// TIA Portal V17 export
// export: Created 2023-02-14T02:49:13.310207Z, ExportSetting WithDefaults, DisplayName Totally Integrated Automation Portal, DisplayVersion V17, DisplayName TIA Portal Openness, DisplayVersion V17, DisplayName TIA Portal Teamcenter Gateway, DisplayVersion V17, DisplayName TIA Portal Version Control Interface, DisplayVersion V17, DisplayName SINAMICS Startdrive Advanced, DisplayVersion V17, DisplayName SINAMICS Startdrive G130, G150, S120, S150, SINAMICS MV, S210, DisplayVersion V17, DisplayName SINAMICS Startdrive G110M, G120, G120C, G120D, G120P, G115D, DisplayVersion V17, DisplayName STEP 7 Professional, DisplayVersion V17, DisplayName STEP 7 Safety, DisplayVersion V17, DisplayName WinCC Professional, DisplayVersion V17
DATA_BLOCK "Mix_to_Salt"   // DB20
{ S7_Optimized_Access := 'FALSE' }
VERSION : 0.1
// stored: AutoNumber false, DBAccessibleFromOPCUA true, DBAccessibleFromWebserver true, IsOnlyStoredInLoadMemory false, IsWriteProtectedInAS false
   VAR
      Heartbeat : Bool;   // Alternating value of 0 and 1 to indicate that the PLC is alive
      Salt_Request : Bool;   // Customer calling for filling to mixer. Batching process will start after receive this signal
      Mixer_TankNum : Int;   // Customer to specify which mixer the transfer will go to (integer value 1 to 12 for mixer 1 to 12)
      "Weight SP" : Real;   // Customer to specify the total weight to batch
   END_VAR
BEGIN
END_DATA_BLOCK
